{attribute 'GeneratedUsingTerminal: EJ1122-0000-0016'}
{attribute addProperty BoxType "EJ1122-0000-0016"}
{attribute addProperty Id "EtcSlaveTerminalBaseInfoDataAT %I*InfoData_6F19DB2B2"}
{attribute addProperty CRC "2874840167"}
{attribute addProperty Size "2"}
TYPE EJ1122_AB5A9467 EXTENDS EtcSlaveTerminalBase :
STRUCT
	{attribute addProperty Name "InfoData"}
	InfoData : InfoData_6F19DB2B;
END_STRUCT
END_TYPE

(* stored: Version 1.2.0.0, ProductVersion 3.1.4024.9
   DUT EJ1122_AB5A9467: Id {bea739f1-451e-49ae-9782-44fb955fc95d} *)
